ABB RobotStudio station: MPS_2025_26_4AHET_ROBOT.rsstnx

Station MPS_2025_26_4AHET_ROBOT (saved by RobotStudio 25.1.11167.1)
Controller IRB120_3_58, task T_ROB1: task frame (RAPID world) sits at (600, 0, 760) mm, rotated rx 0 ry 0 rz 180 deg in the station
Controller IRB120_3_58
  mechanical unit ROB_1: IRB120_3_58__01, 6 joints, base frame (0, 0, 0) mm
Layout (positions relative to the parent item):
  - IRB120_3_58__01 [mechanism, from %ABB.RobotStudio.Models.IRB120%\IRB120_3_58_G_01.rslib] at (600, 0, 760) mm, rotated rx 0 ry 0 rz 180 deg; joint values [0, 0, 0, 0, 0.5236, 0] (rad or m)
  - GENERIC_MPS [part] at (0, 0, 760) mm, size 736.7 x 352.1 x 821.3 mm
  - SCHUNK 40mm Gripper [mechanism, from Components\SCHUNK 40mm Gripper.rslib] at (235.65, 0, 1354) mm, rotated rx -90 ry 60 rz 0 deg
  - GENERIC_MPS_2 [part] at (0, 350, 760) mm, size 736.7 x 352.1 x 821.3 mm
  - GENERIC_MPS_3 [part] at (0, -350, 760) mm, size 736.7 x 352.1 x 821.3 mm
Attachment: SCHUNK 40mm Gripper is attached to IRB120_3_58__01 / Link6
Targets, tools, work objects and paths stored in the station, written as RAPID:
! task T_ROB1
MODULE CalibData
  PERS tooldata MyTool:=[TRUE,[[31.792631019,0,229.638935148],[0.945518576,0,0.325568154,0]],[1,[0,0,1],[1,0,0,0],0,0,0]];
  PERS tooldata schunk_gripper:=[TRUE,[[0,0,0],[0.707106781,0,0.707106781,0]],[1,[0,0,1],[1,0,0,0],0,0,0]];
ENDMODULE

